// TIA Portal project "PID_EPICS_v4" (V15)

(* hardware
DEVICE "S71500/ET200MP station_1"  S7-1500 station
   slot 0: "Rail_0"  Rack  6ES7 590-1***0-0AA0
   slot 1: "PLC_1"  CPU 1516-3 PN/DP  6ES7 516-3AN01-0AB0  V2.5
      slot 3: "CPU display_1"  6ES7591-1BA00-0AA0
*)

// ===== PLC "PLC_1"  CPU 1516-3 PN/DP =====

VAR_GLOBAL   // PLC tag table "UNICOS Tags"
   "T_CYCLE" AT %MD100 : Time;   // Cyclic Time of OB1
   "PID_EXEC_CYCLE" AT %MD104 : Time;   // Cyclic Time of calling all controllers
   "comm" AT %M108.0 : Bool;   // = 1 when FC_event is called
   "UNICOS_LiveCounter" AT %MD110 : DInt;   // Live Counter icncremented each 1 second
   "UNICOS_TimeSmooth" AT %MW114 : Int;   // TimeSmoothing for alarms (user)
   "UNICOS_Counter1" AT %MW116 : Int;   // Counter of PLC sampling til 1 second
   "First_Cycle" AT %M118.0 : Bool;   // Bit to identify the first cycle in the PLC
END_VAR

TYPE "AA_ManRequest"
TITLE = AA_ManRequest
// parameters of Analog Objects
   STRUCT
      ManReg01 : Word;
      HH : Real;
      H : Real;
      L : Real;
      LL : Real;
   END_STRUCT;
END_TYPE

TYPE "AA_bin_Status"
TITLE = AA_bin_Status
// parameters of Analog Objects
   STRUCT
      StsReg01 : Word;
      StsReg02 : Word;
   END_STRUCT;
END_TYPE

TYPE "AA_ana_Status"
TITLE = AA_ana_Status
// parameters of Analog Objects
   STRUCT
      PosSt : Real;
      HHSt : Real;
      HSt : Real;
      LSt : Real;
      LLSt : Real;
   END_STRUCT;
END_TYPE

TYPE "AA_event"
TITLE = AA_event
// parameters of AA Objects
   STRUCT
      evStsReg01 : DWord;
      evStsReg02 : DWord;
   END_STRUCT;
END_TYPE

TYPE "CPC_DB_PA_STATUS"
TITLE = 'CPC_DB_PA_STATUS'
// AFIC Framework
//  Created by GTD based on UNICOS http://unicos.web.cern.ch/
//  DATA STRUCTURES ******************************************************************************
   STRUCT
      ReadBack : Real;   // position of the valve
      ReadBack_status : Byte;   // status of readback
      Pos_D : Byte;   // position discrete
      Pos_D_Status : Byte;   // status of Pos_D
      CheckBack0 : Byte;   // checkback status 0
      CheckBack1 : Byte;   // checkback status 1
      CheckBack2 : Byte;   // checkback status 2
   END_STRUCT;
END_TYPE

TYPE "CPC_DB_COMM"
TITLE = 'CPC_DB_COMM'
// Type for the communication DB
   STRUCT
      status_DB : Int;
      status_DB_old : Int;
      size : Int;
   END_STRUCT;
END_TYPE

TYPE "CPC_ONOFF_PARAM"
TITLE = 'CPC_ONOFF_PARAM'
// Parameters of ONOFF
   STRUCT
      ParReg : Word;
      PPulseLe : Time;
      PWDt : Time;
   END_STRUCT;
END_TYPE

TYPE "CPC_LOCAL_PARAM"
TITLE = 'CPC_LOCAL_PARAM'
// Parameters of LOCAL
   STRUCT
      ParReg : Word;
   END_STRUCT;
END_TYPE

TYPE "CPC_ANALOGALARM_PARAM"
TITLE = 'CPC_ANALOGALARM_PARAM'
// Parameters of Analog Alarm
   STRUCT
      ParReg : Word;
   END_STRUCT;
END_TYPE

TYPE "CPC_PCO_PARAM"
TITLE = 'CPC_PCO_PARAM'
// Parameters of PCO
   STRUCT
      ParReg : Word;
   END_STRUCT;
END_TYPE

TYPE "CPC_ANALOG_PARAM"
TITLE = 'CPC_ANALOG_PARAM'
// Parameters of Analog and Anadig Objects
   STRUCT
      ParReg : Word;
      PMaxRan : Real;
      PMinRan : Real;
      PMStpInV : Real;
      PMStpDeV : Real;
      PMInSpd : Real;
      PMDeSpd : Real;
      PWDt : Time;
      PWDb : Real;
   END_STRUCT;
END_TYPE

TYPE "CPC_STPMOT_PARAM"
TITLE = 'CPC_STPMOT_PARAM'
// Parameter of Stepping Motor Objects
   STRUCT
      ParReg : Word;
      PRefPos : Real;
      PMinRan : Real;
      PMaxRan : Real;
      PSca : Real;
      POffset : Real;
      PMaxSpd : Int;
      PWDt : Time;
      PWDb : Real;
      PDbT : Real;
   END_STRUCT;
END_TYPE

TYPE "CPC_ANADIG_PWM_PARAM"
TITLE = 'PARAM_PWM'
// Parameters of the Pulse Wave Modulation of Anadig objects
   STRUCT
      PTPeriod : Time;
      PTMin : Time;
      PInMax : Real;
   END_STRUCT;
END_TYPE

TYPE "CPC_PID_LIB_PARAM"
TITLE = 'PARAM_PID_LIB'
// Parameters of the PID
   STRUCT
      Kc : Real;
      Ti : Real;
      Td : Real;
      Tds : Real;
      SPH : Real;
      SPL : Real;
      OutH : Real;
      OutL : Real;
      EKc : Bool;
      ETi : Bool;
      ETd : Bool;
      ETds : Bool;
      ESPH : Bool;
      ESPL : Bool;
      EOutH : Bool;
      EOutL : Bool;
   END_STRUCT;
END_TYPE

TYPE "CPC_PID_PARAM"
TITLE = 'PARAM_PID'
// Parameters of controller objects
   STRUCT
      PMinRan : Real;
      PMaxRan : Real;
      POutMinRan : Real;
      POutMaxRan : Real;
      MVFiltTime : Time;
      PIDCycle : Time;
      ScaMethod : Int;
      RA : Bool;
   END_STRUCT;
END_TYPE

TYPE "CPC_RAMP_PARAM"
TITLE = 'PARAM_RAMP'
// Ramp parameters for PID
   STRUCT
      InSpd : Real;
      DeSpd : Real;
   END_STRUCT;
END_TYPE

TYPE "CPC_IOERROR"
TITLE = 'TYPE_ERR'
// Used for IOError in AI/DI/AO/DO
   STRUCT
      ADDR : Real;   // Channel Adress
      Err : Bool;   // Error
   END_STRUCT;
END_TYPE

TYPE "FOF"
TITLE = 'TYPE_FOF'
// Parameters of First Order Filter in Analog Inputs
   STRUCT
      FilterTime : Real;
      Output_old : Real;
   END_STRUCT;
END_TYPE

TYPE "CPC_DB_AA"
TITLE = 'CPC_DB_AA'
// AFIC Framework
//  Created by GTD based on UNICOS http://unicos.web.cern.ch/
//  ANALOG ALARM OBJECT DATA STRUCTURE ****************
   STRUCT
      I : Real;
      PosSt : Real;
      HHSt : Real;
      HSt : Real;
      LSt : Real;
      LLSt : Real;
      HH : Real;
      H : Real;
      L : Real;
      LL : Real;
      PAlDt : Int;
      index : Int;
      PAA : "CPC_ANALOGALARM_PARAM";
      AuAlAck : Bool;
      ISt : Bool;
      WSt : Bool;
      AlUnAck : Bool;
      MAlBRSt : Bool;
      AuIhMB : Bool;
      IOErrorW : Bool;
      IOSimuW : Bool;
      IOError : Bool;
      IOSimu : Bool;
      AuEHH : Bool;
      AuEH : Bool;
      AuEL : Bool;
      AuELL : Bool;
      HHAlSt : Bool;
      HWSt : Bool;
      LWSt : Bool;
      LLAlSt : Bool;
      ConfigW : Bool;
      EHHSt : Bool;
      EHSt : Bool;
      ELSt : Bool;
      ELLSt : Bool;
      ArmRcpSt : Bool;
      PAuAckAl : Bool;
      RemLocSt : Bool;   // 0=Remote, 1=Local Old values Kept
      MAlBSetRst_old : Bool;
      MAlAck_old : Bool;
      AuAlAck_old : Bool;
      Alarm_Cond_old : Bool;
      MNewHHR_old : Bool;
      MNewHR_old : Bool;
      MNewLR_old : Bool;
      MNewLLR_old : Bool;
      ArmRcp_old : Bool;
      ActRcp_old : Bool;
      AlUnAck_old : Bool;   // Delayed properties
      HH_AlarmPh1 : Bool;
      HH_AlarmPh2 : Bool;
      H_AlarmPh1 : Bool;
      H_AlarmPh2 : Bool;
      L_AlarmPh1 : Bool;
      L_AlarmPh2 : Bool;
      LL_AlarmPh1 : Bool;
      LL_AlarmPh2 : Bool;
      HH_TimeAlarm : DInt;
      H_TimeAlarm : DInt;
      L_TimeAlarm : DInt;
      LL_TimeAlarm : DInt;
      TimeAlarm : DInt;
      Iinc : Int;
      Winc : Int;
      HHinc : Int;
      Hinc : Int;
      Linc : Int;
      LLinc : Int;
      WISt : Bool;
      WWSt : Bool;
      WHHAlSt : Bool;
      WHWSt : Bool;
      WLWSt : Bool;
      WLLAlSt : Bool;   // GTD modified
      IhMHHSt : Bool;
      IhMHSt : Bool;
      IhMLSt : Bool;
      IhMLLSt : Bool;
      PosHHW : Bool;   // Threshold Sub-Alarms
      PosHW : Bool;
      PosLW : Bool;
      PosLLW : Bool;
   END_STRUCT;
END_TYPE

TYPE "CPC_DB_AI"
TITLE = 'CPC_DB_AI'
// AFIC Framework
//  Created by GTD based on UNICOS http://unicos.web.cern.ch/
//  ANALOG INPUT OBJECT DATA STRUCTURE *************************
   STRUCT
      perAddress : Int;   // Input periphery address
      FEType : Int;   // Type of AI (0-> Direct address, 2-> Sipart Profibus PA)
      index : Int;   // Index of the AI (recognize its status position)
      HFPos : Int;   // Value from periphery (INTEGER)
      PMinRan : Real;   // Range Min
      PMaxRan : Real;   // Range Max
      PMinRaw : Int;   // Raw Min
      PMaxRaw : Int;   // Raw Max
      PDb : Real;   // Dead Band
      PosSt : Real;   // Position Status
      HFSt : Real;   // Hardware Position Status
      MPosRSt : Real;   // Manual Position Request Status
      Autoi_old : Real;
      MNewMR_old : Bool;
      AuIhFoMo : Bool;   // Forced mode inhibited by logic
      AuMoSt : Bool;   // Auto Mode status (StsReg01 bit 2)
      FoMoSt : Bool;   // Force Mode status (StsReg01 bit 4)
      IOErrorW : Bool;   // Error in input (StsReg01 bit 6)
      IOSimuW : Bool;   // Input simulated (StsReg01 bit 7)
      IOError : Bool;
      IOSimu : Bool;
      FoDiProW : Bool;   // Forced Mode-Process discordance (StsReg01 bit 8)
      PiwDef : Bool;   // PIW definition (true) or IW definition (false)
      MIOErBRSt : Bool;   // Manual IOError Block Request Status
      MIOErBSetRst_old : Bool;   // Manual IOError Block Set/Reset Old value
      FOFEn : Bool;   // First Order Filter Enabling Bit
      RemLocSt : Bool;   // 0=Remote, 1=Local
      IOErrReact : Bool;   // IO Error Reaction (0=Go to default value, 1=Keep last known value)
   END_STRUCT;
END_TYPE

TYPE "CPC_DB_AIR"
TITLE = 'CPC_DB_AIR'
// AFIC Framework
//  Created by GTD based on UNICOS http://unicos.web.cern.ch/
//  ANALOG INPUT REAL OBJECT DATA STRUCTURE *************************
   STRUCT
      FEType : Int;   // (0-> no addressing, 1-> DB addresss, 2-> type 1 + DB adress Ioerror)
      DBnum : Int;   // Front End Type InterfaceParam1. Db number (i.e.: 10 -> DB10)
      DBpos : Int;   // Front End Type InterfaceParam2. Db position (i.e: 20 -> DBxx.DBD20)
      DBnumIoError : Int;   // Front End Type InterfaceParam3. Db number (i.e.: 10 -> DB10
      DBposIoError : Int;   // Front End Type InterfaceParam4. Db position (i.e: 20 -> DBxx.DBD20.y)
      DBbitIoError : Int;   // Front End Type InterfaceParam5. Db bit (i.e: 5 -> DBxx.DBD20.5)
      index : Int;   // Index of the AIC (recognize its status position)
      HFPos : Real;   // Value from (REAL)
      PMinRan : Real;   // Range Min
      PMaxRan : Real;   // Range Max
      PMinRaw : Real;   // Scale Min
      PMaxRaw : Real;   // Scale Max
      PDb : Real;   // Dead Band
      MPosRSt : Real;   // Manual Position Request Status
      PosSt : Real;   // Position Status
      HFSt : Real;   // Hardware Position Status
      Autoi_old : Real;
      MNewMR_old : Bool;
      AuIhFoMo : Bool;   // Force mode blocked by logic
      AuMoSt : Bool;   // Auto Mode status (StsReg01 bit=2)
      FoMoSt : Bool;   // Force Mode status (StsReg01 bit 4)
      IOErrorW : Bool;   // Error in input (StsReg01 bit 6)
      IOSimuW : Bool;   // Input simulated (StsReg01 bit 7)
      IOError : Bool;
      IOSimu : Bool;
      FoDiProW : Bool;   // Forced discordance (StsReg01 bit 8)
      MIOErBRSt : Bool;   // Manual IOError Block Request Status
      MIOErBSetRst_old : Bool;   // Manual IOError Block Request Set/Reset old value
      PIWDef : Bool;
      FOFEn : Bool;   // First Order Filter Enabling Bit
      RemLocSt : Bool;   // 0=Remote, 1=Local
      IOErrReact : Bool;   // IO Error Reaction (0=Go to default value, 1=Keep last known value)
   END_STRUCT;
END_TYPE

TYPE "CPC_DB_AO"
TITLE = 'CPC_DB_AO'
// AFIC Framework
//  Created by GTD based on UNICOS http://unicos.web.cern.ch/
//  ANALOG OUTPUT OBJECT DATA STRUCTURE *************************
   STRUCT
      perAddress : Int;   // Input periphery address
      FEType : Int;
      index : Int;   // Index of the AO (recognize its status position)
      AuPosR : Real;   // Real value
      PMinRan : Real;   // Range Min
      PMaxRan : Real;   // Range Max
      PMinRaw : Int;   // Scale Min
      PMaxRaw : Int;   // Scale Max
      PosSt : Real;   // Status (real value)
      MPosRSt : Real;   // Manual Position Request Status
      AuPosRSt : Real;   // Auto Position Request Status
      OutOV : Int;   // Output order
      AuIhFoMo : Bool;   // Force mode blocked by logic (StsReg01 bit=13)
      AuMoSt : Bool;   // Auto Mode status (StsReg01 bit=2)
      FoMoSt : Bool;   // Force Mode status (StsReg01 bit 4)
      IOErrorW : Bool;   // Error in input (StsReg01 bit 6)
      IOSimuW : Bool;   // Input simulated (StsReg01 bit 7)
      IOError : Bool;
      IOSimu : Bool;
      FoDiAuW : Bool;   // Forced discordance (StsReg01 bit 8)
      PqwDef : Bool;   // PQW definition (true) or QW definition (false)
      MIOErBRSt : Bool;   // Manual IOError Block Request Status
      MIOErBSetRst_old : Bool;   // Manual IOError Block Set/Reset old value
      MNewMR_old : Bool;
      RemLocSt : Bool;   // 0=Remote, 1=Local
   END_STRUCT;
END_TYPE

TYPE "CPC_DB_AOR"
TITLE = 'CPC_DB_AOR'
// AFIC Framework
//  Created by GTD based on UNICOS http://unicos.web.cern.ch/
//  ANALOG OUTPUT REAL OBJECT DATA STRUCTURE *************************
   STRUCT
      FEType : Int;
      index : Int;   // Index of the AOC (recognize its status position)
      DBnum : Int;   // Db number (i.e.: 10 -> DB10)
      DBpos : Int;   // Db position (i.e: 20 -> DBxx.DBD20)
      DBnumIoError : Int;   // Db number (i.e.: 10 -> DB10
      DBposIoError : Int;   // Db position (i.e: 20 -> DBxx.DBD20.y)
      DBbitIoError : Int;   // Db bit (i.e: 5 -> DBxx.DBD20.5)
      AuPosR : Real;   // Real value
      PMinRan : Real;   // Range Min
      PMaxRan : Real;   // Range Max
      PMinRaw : Real;   // Row Min
      PMaxRaw : Real;   // Row Max
      PosSt : Real;   // Status (real value)
      OutOV : Real;   // Output order
      MPosRSt : Real;   // Manual Position Request Status
      AuPosRSt : Real;   // Auto Position Request Status
      MNewMR_old : Bool;
      AuIhFoMo : Bool;   // Force mode blocked by logic (StsReg01 bit=13)
      AuMoSt : Bool;   // Auto Mode status (StsReg01 bit=2)
      FoMoSt : Bool;   // Force Mode status (StsReg01 bit 4)
      IOErrorW : Bool;   // Error in input (StsReg01 bit 6)
      IOSimuW : Bool;   // Input simulated (StsReg01 bit 7)
      IOError : Bool;
      IOSimu : Bool;
      AuMRW : Bool;   // Forced discordance (StsReg01 bit 8)
      MIOErBRSt : Bool;   // Manual IOError Block Request Status
      MIOErBSetRst_old : Bool;   // Manual IOError Block Set/Reset Old value
      PQWDef : Bool;
      RemLocSt : Bool;   // 0=Remote, 1=Local
   END_STRUCT;
END_TYPE

TYPE "CPC_DB_APAR"
TITLE = 'CPC_DB_APAR'
// AFIC Framework
//  Created by GTD based on UNICOS http://unicos.web.cern.ch/
//  ANALOG PARAMETER OBJECT DATA STRUCTURE *************************
   STRUCT
      PosSt : Real;
      MPosRSt : Real;
      ArmRcp_old : Bool;
      ActRcp_old : Bool;
      MNewMR_old : Bool;
      ArmRcpSt : Bool;
      index : Int;   // Index within the arrays
      RemLocSt : Bool;   // 0=Remote, 1=Local
   END_STRUCT;
END_TYPE

TYPE "CPC_DB_AS"
TITLE = 'CPC_DB_AS'
// AFIC Framework
//  Created by GTD based on UNICOS http://unicos.web.cern.ch/
//  ANALOG STATUS OBJECT DATA STRUCTURE *************************
   STRUCT
      index : Int;   // Index of the AI (recognize its status position)
      FEType : Int;
      InterfaceParam1 : Int;   // Input periphery address
      InterfaceParam2 : Int;   // Input periphery address
      AuPosR : Real;
      PosSt : Real;
      PIWDef : Bool;
      FOFEn : Bool;   // First Order Filter Enabling Bit
   END_STRUCT;
END_TYPE

TYPE "CPC_DB_DA"
TITLE = 'CPC_DB_DA'
// AFIC Framework
//  Created by GTD based on UNICOS http://unicos.web.cern.ch/
//  DIGITAL ALARM OBJECT DATA STRUCTURE ****************
   STRUCT
      PAlDt : Int;
      index : Int;
      PAuAckAl : Bool;
      I : Bool;
      AuAlAck : Bool;
      ISt : Bool;
      AlUnAck : Bool;
      MAlBRSt : Bool;
      AuIhMB : Bool;
      IOErrorW : Bool;
      IOSimuW : Bool;
      IOError : Bool;
      IOSimu : Bool;
      AuEAl : Bool := TRUE;
      RemLocSt : Bool;   // 0=Remote; 1=Local
      MAlBSetRst_old : Bool;   // Old values Kept
      MAlAck_old : Bool;
      AuAlAck_old : Bool;
      Alarm_Cond_old : Bool;
      AlUnAck_old : Bool;
      AlarmPh1 : Bool;   // Delayed properties
      AlarmPh2 : Bool;
      WISt : Bool;
      TimeAlarm : DInt;
      Iinc : Int;   // GTD modified
      PosW : Bool;
      ConfigW : Bool;
   END_STRUCT;
END_TYPE

TYPE "CPC_DB_DI"
TITLE = 'CPC_DB_DI'
// AFIC Framework
//  Created by GTD based on UNICOS http://unicos.web.cern.ch/
//  DIGITAL INPUT OBJECT DATA STRUCTURE ****************
   STRUCT
      FEType : Int;   // Type of AI (0-> Direct address, 2-> Sipart Profibus PA)
      index : Int;   // Index of the AI (recognize its status position)
      DBnum : Int;
      perByte : Int;
      perBit : Int;
      DBnumIoError : Int;
      DBposIoError : Int;
      DBbitIoError : Int;
      AuIhFoMo : Bool;   // Forced mode inhibited by logic
      PosSt : Bool;   // Position Status
      MPosRSt : Bool;   // Manual Position Request Status
      HFSt : Bool;   // Hardware Position Status
      AuMoSt : Bool;   // Auto Mode status
      FoMoSt : Bool;   // Force Mode status
      IOErrorW : Bool;   // Error in input
      IOSimuW : Bool;   // Input simulated
      IOError : Bool;
      IOSimu : Bool;
      FoDiProW : Bool;   // Forced Mode-Process discordance
      HFPos : Bool;   // Value from periphery (BOOL)
      MIOErBRSt : Bool;   // Manual IOError Block Request Status
      MIOErBSetRst_old : Bool;   // Manual IOError Block Set/Reset Old value
      RemLocSt : Bool;   // 0=Remote, 1=Local
      IOErrReact : Bool;   // IO Error Reaction (0=Go to default value, 1=Keep last known value)
   END_STRUCT;
END_TYPE

TYPE "CPC_DB_DO"
TITLE = 'CPC_DB_DO'
// AFIC Framework
//  Created by GTD based on UNICOS http://unicos.web.cern.ch/
//  DIGITAL OUTPUT OBJECT DATA STRUCTURE ****************
   STRUCT
      FEType : Int;
      index : Int;
      DBnum : Int;
      perByte : Int;
      perBit : Int;
      DBnumIoError : Int;
      DBposIoError : Int;
      DBbitIoError : Int;
      AuIhFoMo : Bool;
      PosSt : Bool;
      MPosRSt : Bool;
      AuPosRSt : Bool;
      AuMoSt : Bool;
      FoMoSt : Bool;
      IOErrorW : Bool;
      IOSimuW : Bool;
      IOError : Bool;
      IOSimu : Bool;
      FoDiAuW : Bool;
      AuPosR : Bool;
      MIOErBRSt : Bool;
      MIOErBSetRst_old : Bool;
      RemLocSt : Bool;   // 0= Remote, 1=Local
   END_STRUCT;
END_TYPE

TYPE "CPC_DB_DPAR"
TITLE = 'CPC_DB_DPAR'
// AFIC Framework
//  Created by GTD based on UNICOS http://unicos.web.cern.ch/
//  DIGITAL PARAMETER OBJECT DATA STRUCTURE ****************
   STRUCT
      PosSt : Bool;
      ArmRcp_old : Bool;
      ActRcp_old : Bool;
      MOnR_old : Bool;
      MOffR_old : Bool;
      ArmRcpSt : Bool;
      MOnRSt : Bool;
      MOffRSt : Bool;
      RemLocSt : Bool;   // 0 =Remote, 1=Local
      index : Int;   // Index for identification
   END_STRUCT;
END_TYPE

TYPE "CPC_DB_ENC"
TITLE = 'CPC_DB_ENC'
// AFIC Framework
//  Created by GTD based on UNICOS http://unicos.web.cern.ch/
//  ENCODER OBJECT DATA STRUCTURE *************************
   STRUCT
      perAddress : Int;   // Input periphery address
      FEType : Int;   // Type of ADDRESSING
      PEType : Int;   // Type of ENCODER
      index : Int;   // Index of the ENC
      HFPos : DWord;   // Value from periphery (DWORD)
      PMinRan : Real;   // Range Min
      PMaxRan : Real;   // Range Max
      PMinRaw : Int;   // Raw Min
      PMaxRaw : Int;   // Raw Max
      PDb : Real;   // Dead Band
      PosSt : Real;   // Position Status
      HFSt : Real;   // Hardware Position Status
      MPosRSt : Real;   // Manual Position Request Status
      Autoi_old : Real;
      MNewMR_old : Bool;
      AuIhFoMo : Bool;   // Forced mode inhibited by logic
      AuMoSt : Bool;   // Auto Mode status (StsReg01 bit 2)
      FoMoSt : Bool;   // Force Mode status (StsReg01 bit 4)
      IOErrorW : Bool;   // Error in input (StsReg01 bit 6)
      IOSimuW : Bool;   // Input simulated (StsReg01 bit 7)
      IOError : Bool;
      IOSimu : Bool;
      FoDiProW : Bool;   // Forced Mode-Process discordance (StsReg01 bit 8)
      PiwDef : Bool;   // PIW definition (true) or IW definition (false)
      MIOErBRSt : Bool;   // Manual IOError Block Request Status
      MIOErBSetRst_old : Bool;   // Manual IOError Block Set/Reset Old value
   END_STRUCT;
END_TYPE

TYPE "CPC_DB_WPAR"
TITLE = 'CPC_DB_WPAR'
// AFIC Framework
//  Created by GTD based on UNICOS http://unicos.web.cern.ch/
//  WORD PARAMETER OBJECT DATA STRUCTURE *************************
   STRUCT
      InterfaceParam1 : Int;   // Input periphery address
      InterfaceParam2 : Int;   // Input periphery address
      FEType : Int;
      index : Int;   // Index of the AI (recognize its status position)
      PosSt : Word;
      MPosRSt : Word;
      RemLocSt : Bool;   // 0=Rmeote, 1=Local
      ArmRcp_old : Bool;
      ActRcp_old : Bool;
      MNewMR_old : Bool;
      ArmRcpSt : Bool;
      PQWDef : Bool;
   END_STRUCT;
END_TYPE

TYPE "CPC_DB_WS"
TITLE = 'CPC_DB_WS'
// AFIC Framework
//  Created by GTD based on UNICOS http://unicos.web.cern.ch/
//  WORD STATUS OBJECT DATA STRUCTURE *************************
   STRUCT
      PIWDef : Bool;
      ReadByte : Bool;
      index : Int;
      FEType : Int;
      InterfaceParam1 : Int;
      InterfaceParam2 : Int;
      AuPosR : Word;
      PosSt : Word;
   END_STRUCT;
END_TYPE

TYPE "AI_ManRequest"
TITLE = AI_ManRequest
// parameters of Analog Objects
   STRUCT
      ManReg01 : Word;
      MPosR : Real;
   END_STRUCT;
END_TYPE

TYPE "AI_bin_Status"
TITLE = AI_bin_Status
// parameters of Analog Objects
   STRUCT
      StsReg01 : Word;
   END_STRUCT;
END_TYPE

TYPE "AI_event"
TITLE = AI_event
// parameters of AI Objects
   STRUCT
      evStsReg01 : DWord;
   END_STRUCT;
END_TYPE

TYPE "AI_ana_Status"
TITLE = AI_ana_Status
// parameters of Analog Objects
   STRUCT
      PosSt : Real;
      HFSt : Real;
   END_STRUCT;
END_TYPE

TYPE "AIR_ManRequest"
TITLE = AIR_ManRequest
// parameters of Analog Objects
   STRUCT
      ManReg01 : Word;
      MPosR : Real;
   END_STRUCT;
END_TYPE

TYPE "AIR_bin_Status"
TITLE = AIR_bin_Status
// parameters of Analog Objects
   STRUCT
      StsReg01 : Word;
   END_STRUCT;
END_TYPE

TYPE "AIR_event"
TITLE = AIR_event
// parameters of ANADIG Objects
   STRUCT
      evStsReg01 : DWord;
   END_STRUCT;
END_TYPE

TYPE "AIR_ana_Status"
TITLE = AIR_ana_Status
// parameters of Analog Objects
   STRUCT
      PosSt : Real;
      HFSt : Real;
   END_STRUCT;
END_TYPE

TYPE "AO_ManRequest"
TITLE = AO_ManRequest
// parameters of Analog Objects
   STRUCT
      ManReg01 : Word;
      MPosR : Real;
   END_STRUCT;
END_TYPE

TYPE "AO_bin_Status"
TITLE = AO_bin_Status
// parameters of Analog Objects
   STRUCT
      StsReg01 : Word;
   END_STRUCT;
END_TYPE

TYPE "AO_event"
TITLE = AO_event
// parameters of Analog Objects
   STRUCT
      evStsReg01 : DWord;
   END_STRUCT;
END_TYPE

TYPE "AO_ana_Status"
TITLE = AO_ana_Status
// parameters of Analog Objects
   STRUCT
      PosSt : Real;
      AuPosRSt : Real;
   END_STRUCT;
END_TYPE

TYPE "AOR_ManRequest"
TITLE = AOR_ManRequest
// parameters of Analog Objects
   STRUCT
      ManReg01 : Word;
      MPosR : Real;
   END_STRUCT;
END_TYPE

TYPE "AOR_bin_Status"
TITLE = AOR_bin_Status
// parameters of Analog Objects
   STRUCT
      StsReg01 : Word;
   END_STRUCT;
END_TYPE

TYPE "AOR_event"
TITLE = AOR_event
// parameters of ANADIG Objects
   STRUCT
      evStsReg01 : DWord;
   END_STRUCT;
END_TYPE

TYPE "AOR_ana_Status"
TITLE = AOR_ana_Status
// parameters of Analog Objects
   STRUCT
      PosSt : Real;
      AuPosRSt : Real;
   END_STRUCT;
END_TYPE

TYPE "APAR_ManRequest"
TITLE = APAR_ManRequest
// parameters of Analog Objects
   STRUCT
      ManReg01 : Word;
      MPosR : Real;
   END_STRUCT;
END_TYPE

TYPE "APAR_bin_Status"
TITLE = APAR_bin_Status
// parameters of Analog Objects
   STRUCT
      StsReg01 : Word;
   END_STRUCT;
END_TYPE

TYPE "APAR_ana_Status"
TITLE = APAR_ana_Status
// parameters of Analog Objects
   STRUCT
      PosSt : Real;
      MPosRSt : Real;
   END_STRUCT;
END_TYPE

TYPE "APAR_event"
TITLE = APAR_event
// parameters of ANADIG Objects
   STRUCT
      evStsReg01 : DWord;
   END_STRUCT;
END_TYPE

TYPE "AS_ana_Status"
TITLE = AS_ana_Status
// parameters of Analog Objects
   STRUCT
      PosSt : Real;
   END_STRUCT;
END_TYPE

TYPE "DA_ManRequest"
TITLE = DA_ManRequest
// parameters of Analog Objects
   STRUCT
      ManReg01 : Word;
   END_STRUCT;
END_TYPE

TYPE "DA_bin_Status"
TITLE = DA_bin_Status
// parameters of DA Objects
   STRUCT
      StsReg01 : Word;
   END_STRUCT;
END_TYPE

TYPE "DA_event"
TITLE = DA_event
// parameters of DA Objects
   STRUCT
      evStsReg01 : DWord;
   END_STRUCT;
END_TYPE

TYPE "DI_ManRequest"
TITLE = DI_ManRequest
// parameters of Analog Objects
   STRUCT
      ManReg01 : Word;
   END_STRUCT;
END_TYPE

TYPE "DI_bin_Status"
TITLE = DI_bin_Status
// parameters of Analog Objects
   STRUCT
      StsReg01 : Word;
   END_STRUCT;
END_TYPE

TYPE "DI_event"
TITLE = DI_event
// parameters of DI Objects
   STRUCT
      evStsReg01 : DWord;
   END_STRUCT;
END_TYPE

TYPE "DO_ManRequest"
TITLE = DO_ManRequest
// parameters of Analog Objects
   STRUCT
      ManReg01 : Word;
   END_STRUCT;
END_TYPE

TYPE "DO_bin_Status"
TITLE = DO_bin_Status
// parameters of Analog Objects
   STRUCT
      StsReg01 : Word;
   END_STRUCT;
END_TYPE

TYPE "DO_event"
TITLE = DO_event
// parameters of AI Objects
   STRUCT
      evStsReg01 : DWord;
   END_STRUCT;
END_TYPE

TYPE "DPAR_ManRequest"
TITLE = DPAR_ManRequest
// parameters of Analog Objects
   STRUCT
      ManReg01 : Word;
   END_STRUCT;
END_TYPE

TYPE "DPAR_bin_Status"
TITLE = DPAR_bin_Status
// parameters of Analog Objects
   STRUCT
      StsReg01 : Word;
   END_STRUCT;
END_TYPE

TYPE "DPAR_event"
TITLE = DPAR_event
// parameters of ANADIG Objects
   STRUCT
      evStsReg01 : DWord;
   END_STRUCT;
END_TYPE

TYPE "ONOFF_ManRequest"
TITLE = ONOFF_ManRequest
// parameters of OnOff Objects
   STRUCT
      ManReg01 : Word;
   END_STRUCT;
END_TYPE

TYPE "ONOFF_bin_Status"
TITLE = ONOFF_bin_Status
// parameters of OnOff Objects
   STRUCT
      StsReg01 : Word;
      StsReg02 : Word;
   END_STRUCT;
END_TYPE

TYPE "ONOFF_event"
TITLE = ONOFF_event
// parameters of OnOff Objects
   STRUCT
      evStsReg01 : DWord;
      evStsReg02 : DWord;
   END_STRUCT;
END_TYPE

TYPE "PCO_ManRequest"
TITLE = PCO_ManRequest
// parameters of Analog Objects
   STRUCT
      ManReg01 : Word;
      MOpMoR : Real;
   END_STRUCT;
END_TYPE

TYPE "PCO_bin_Status"
TITLE = PCO_bin_Status
// parameters of Analog Objects
   STRUCT
      StsReg01 : Word;
      StsReg02 : Word;
   END_STRUCT;
END_TYPE

TYPE "PCO_event"
TITLE = PCO_event
// parameters of AI Objects
   STRUCT
      evStsReg01 : DWord;
      evStsReg02 : DWord;
   END_STRUCT;
END_TYPE

TYPE "PCO_ana_Status"
TITLE = PCO_ana_Status
// parameters of Analog Objects
   STRUCT
      OpMoSt : Real;
      AuOpMoSt : Real;
   END_STRUCT;
END_TYPE

TYPE "WPAR_ManRequest"
TITLE = WPAR_ManRequest
// parameters of Analog Objects
   STRUCT
      ManReg01 : Word;
      MPosR : Word;
   END_STRUCT;
END_TYPE

TYPE "WPAR_bin_Status"
TITLE = WPAR_bin_Status
// parameters of WPAR Objects
   STRUCT
      StsReg01 : Word;
   END_STRUCT;
END_TYPE

TYPE "WPAR_event"
TITLE = WPAR_event
// parameters of WPAR Objects
   STRUCT
      evStsReg01 : DWord;
   END_STRUCT;
END_TYPE

TYPE "WPAR_ana_Status"
TITLE = WPAR_ana_Status
// parameters of Analog Objects
   STRUCT
      PosSt : Word;
      MPosRSt : Word;
   END_STRUCT;
END_TYPE

TYPE "WS_ana_Status"
TITLE = 'WS_ana_Status'
// parameters of Analog Objects
   STRUCT
      PosSt : Word;
   END_STRUCT;
END_TYPE

TYPE "OPC_AI_Status"
   STRUCT
      StsReg01 : Word;
      PosSt : Real;
      HFSt : Real;
   END_STRUCT;
END_TYPE

TYPE "OPC_ONOFF_Status"
   STRUCT
      StsReg01 : Word;
      StsReg02 : Word;
   END_STRUCT;
END_TYPE

TYPE "OPC_PCO_Status"
   STRUCT
      StsReg01 : Word;
      StsReg02 : Word;
      OpMoSt : Real;
      AuOpMoSt : Real;
   END_STRUCT;
END_TYPE

TYPE "OPC_DI_Status"
   STRUCT
      StsReg01 : Word;
   END_STRUCT;
END_TYPE

TYPE "AIR_ManRequest_1"
TITLE = AIR_ManRequest
// parameters of Analog Objects
   STRUCT
      ManReg01 : Bool;
      MPosR : Real;
   END_STRUCT;
END_TYPE

TYPE "WPAR_status"
   STRUCT
      bin_status : "WPAR_bin_Status";
      ana_status : "WPAR_ana_Status";
   END_STRUCT;
END_TYPE

TYPE "AA_status"
   STRUCT
      bin_status : "AA_bin_Status";
      ana_status : "AA_ana_Status";
   END_STRUCT;
END_TYPE

TYPE "AI_status"
   STRUCT
      bin_status : "AI_bin_Status";
      ana_status : "AI_ana_Status";
   END_STRUCT;
END_TYPE

DATA_BLOCK "init"   // DB1
{ S7_Optimized_Access := 'TRUE' }
VERSION : 0.1
   VAR
      St : Real := 0.05;
      kp : Real := 0.91;
      ki : Real := 0.099;
      kd : Real := 0.01;
      SP : Real := 89.0;
      mass : Real := 5.43;
      g : Real := 9.81;
      connreq : Bool;
      sendreq : Bool;
      recreq : Bool;
      discreq : Bool;
   END_VAR
BEGIN
END_DATA_BLOCK

DATA_BLOCK "sendDB"   // DB5
{ S7_Optimized_Access := 'FALSE' }
VERSION : 0.1
   VAR
      St : Real;
      kp : Real;
      ki : Real;
      kd : Real;
      e0 : Real;
      e1 : Real;
      e2 : Real;
      e3 : Real;
      e4 : Real;
      y : Real;
      yout : Real;
   END_VAR
BEGIN
END_DATA_BLOCK

DATA_BLOCK "recDB"   // DB6
{ S7_Optimized_Access := 'FALSE' }
VERSION : 0.1
   VAR
      u4 : Real;
      SP : Real;
   END_VAR
BEGIN
END_DATA_BLOCK

DATA_BLOCK "process"   // DB7
{ S7_Optimized_Access := 'TRUE' }
VERSION : 0.1
   VAR
      y : Real := 1.0;
      e0 : Real := 88.0;
      e1 : Real := 88.0;
      e2 : Real := 88.0;
      e3 : Real := 88.0;
      e4 : Real := 88.0;
      u0 : Real;
      u1 : Real;
      u2 : Real;
      u3 : Real;
      u4 : Real;
   END_VAR
BEGIN
END_DATA_BLOCK

DATA_BLOCK "testDB"   // DB10
{ S7_Optimized_Access := 'FALSE' }
VERSION : 0.1
   VAR
      testSend : Real;
      epicsu4 : Real;
      SP : Real;
   END_VAR
BEGIN
END_DATA_BLOCK

// folder: System blocks/Program resources

DATA_BLOCK "PLC_1_Connection_DB"   // DB3
{ S7_Optimized_Access := 'TRUE' }
AUTHOR : SIMATIC
FAMILY : MC7Plus
NAME : TC_IP_v4
VERSION : 1.0
// stored: InstanceOfName TCON_IP_v4
"TCON_IP_v4"
BEGIN
   ID := 1;
   InterfaceId := 64;
   LocalPort := 2000;
END_DATA_BLOCK

// folder: (top level)

FUNCTION "newpos" : Void   // FC1, SCL
{ S7_Optimized_Access := 'TRUE' }
VERSION : 0.1
   VAR_TEMP
      vzero : Real;
      power : Real;
   END_VAR
BEGIN
   IF  "TRCV_DB".NDR THEN

       "process".e0 := "process".e1;
       "process".e1 := "process".e2;
       "process".e2 := "process".e3;
       "process".e3 := "process".e4;
       "process".e4 := "init".SP - "process".y;


       "process".u0 := "process".u1;
       "process".u1 := "process".u2;
       "process".u2 := "process".u3;
       "process".u3 := "process".u4;

        "process".u4 := "recDB".u4;
       // u4 is calculated by epics 

       //"process".u4 := "init".kp * "process".e4 + "init".ki / (5 * "init".St) * ("process".e0 + "process".e1 + "process".e2 + "process".e3 + "process".e4) + ("process".e3 - "process".e4) * "init".kd / "init".St;

       #vzero := ("process".u0 / "init".mass + "process".u1 / "init".mass + "process".u2 / "init".mass + "process".u3 / "init".mass + "process".u4 / "init".mass - 5 * "init".g);
       #power := "init".St * "init".St;
       "process".y := "process".y + #vzero * "init".St + 0.5 * ("process".u4 / "init".mass - "init".g) * #power;


   END_IF;
END_FUNCTION

FUNCTION "tcpServer" : Void   // FC2, SCL
{ S7_Optimized_Access := 'TRUE' }
VERSION : 0.1
BEGIN
   "TCON_DB"(REQ:="init".connreq,
             ID:=1,
             CONNECT:="PLC_1_Connection_DB", DONE => "TCON_DB".DONE, BUSY => "TCON_DB".BUSY, ERROR => "TCON_DB".ERROR, STATUS => "TCON_DB".STATUS);


   "TSEND_DB".TSEND(REQ := "init".sendreq,
                    ID := 1,
                    LEN := 44,
                    DONE => "TSEND_DB".DONE,
                    BUSY => "TSEND_DB".BUSY,
                    ERROR => "TSEND_DB".ERROR,
                    STATUS => "TSEND_DB".STATUS,
                    DATA := "sendDB");

   "TRCV_DB".TRCV(EN_R:="init".recreq,
                  ID:=1,
                  LEN:=8,
                  ADHOC:=0,
                  NDR=>"TRCV_DB".NDR,
                  BUSY=>"TRCV_DB".BUSY,
                  ERROR=>"TRCV_DB".ERROR,
                  STATUS=>"TRCV_DB".STATUS,
                  RCVD_LEN=>"TRCV_DB".RCVD_LEN,
                  DATA:="recDB");

   "TDISCON_DB"(REQ:="init".discreq,
                ID:=1,
                DONE=>"TDISCON_DB".DONE,
                BUSY=>"TDISCON_DB".BUSY,
                ERROR=>"TDISCON_DB".ERROR,
                STATUS=>"TDISCON_DB".STATUS);
END_FUNCTION

FUNCTION "sendmap" : Void   // FC3, SCL
{ S7_Optimized_Access := 'TRUE' }
VERSION : 0.1
BEGIN
   "sendDB".St := "init".St;
   "sendDB".kp := "init".kp;
   "sendDB".ki := "init".ki;
   "sendDB".kd := "init".kd;
   "sendDB".e0 := "process".e0;
   "sendDB".e1 := "process".e1;
   "sendDB".e2 := "process".e2;
   "sendDB".e3 := "process".e3;
   "sendDB".e4 := "process".e4;
   "sendDB".y := "process".y;
   "sendDB".yout := "process".y + 18.43;
END_FUNCTION

FUNCTION "recmap" : Void   // FC4, SCL
{ S7_Optimized_Access := 'TRUE' }
VERSION : 0.1
BEGIN
   //"process".u4 := "recDB".u4;
   "init".SP := "recDB".SP;
   "testDB".epicsu4 := "recDB".u4;
   "testDB".SP := "init".SP;
END_FUNCTION

FUNCTION "connMGM" : Void   // FC5, SCL
{ S7_Optimized_Access := 'TRUE' }
VERSION : 0.1
BEGIN
   IF ("init".connreq = 1  AND "init".sendreq = 0) THEN
       "init".sendreq := 1;
   END_IF;

   IF ("TSEND_DB".DONE = 1 ) THEN
       "init".sendreq := 0;
   END_IF;
END_FUNCTION

ORGANIZATION_BLOCK "Main"   // OB1, STL, ProgramCycle
TITLE = "Main Program Sweep (Cycle)"
{ S7_Optimized_Access := 'FALSE' }
VERSION : 0.1
   VAR_TEMP
      EV_CLASS : Byte;   // Bits 0-3 = 1:Coming event, Bits 4-7 = 1:Event class 1
      SCAN_1 : Byte;   // 1:Initial call of the OB, 3: Call 2-n of the OB
      PRIORITY : Byte;   // Priority of OB Execution
      OB_NUMBR : Byte;   // OB number
      RESERVED_1 : Byte;   // Reserved for system
      RESERVED_2 : Byte;   // Reserved for system
      PREV_CYCLE : Int;   // Previous program cycle time (milliseconds)
      MIN_CYCLE : Int;   // Minimum program cycle time (milliseconds)
      MAX_CYCLE : Int;   // Maximum program cycle time (milliseconds)
      DATE_TIME : Date_And_Time;   // Date and time OB started
   END_VAR
BEGIN

REGION Network 1




         CALL  "newpos";

         CALL  "sendmap";

         CALL  "tcpServer";



         CALL  "connMGM";
         CALL  "recmap";
END_REGION
END_ORGANIZATION_BLOCK